// TIA Portal V20 export
TYPE "LBP_typeMcp310AdditionalOutput"
TITLE = MCP 310 image / Image du MCP 310
// Additional output image of MCP 310 / Image de sortie supplémentaire du MCP 310
   STRUCT
      reserved0 : Byte;
      reserved1 : Byte;
   END_STRUCT;
END_TYPE
